Fanuc KAREL source: CA0044.KL

-- PROVISIONAL review KL for V770-1; original PC SHA256 f519f34b8b673ea591116af9cf0e5e1c5a1d14f930d2b18fb79fd747858d793d
-- Incomplete behavior may be omitted. Consult companion uncertainty JSON. Do not deploy.
PROGRAM CA0044
%NOLOCKGROUP
BEGIN
  -- UNRESOLVED_PC offsets 0-1; opcodes 7B
  -- UNRESOLVED_PC offsets 6-20; opcodes 21,9D,52,23
  -- UNRESOLVED_PC offsets 25-29; opcodes 7F
  -- UNRESOLVED_PC offsets 34-41; opcodes 9C,23
  -- UNRESOLVED_PC offsets 46-53; opcodes 9D,23
  -- UNRESOLVED_PC offsets 58-69; opcodes 2E,23
  -- UNRESOLVED_PC offsets 74-81; opcodes 9D,23
  -- UNRESOLVED_PC offsets 86-95; opcodes 3F,75
  -- UNRESOLVED_PC offsets 100-114; opcodes 2E,22,9D,33,35
  -- UNRESOLVED_PC offsets 119-133; opcodes 2E,22,9D,33,35
  -- UNRESOLVED_PC offsets 138-153; opcodes 2E,22,32,35
  -- UNRESOLVED_PC offsets 158-173; opcodes 2E,22,32,35
  -- UNRESOLVED_PC offsets 178-350; opcodes 27,27,21,27,21,27,21,27,21,27,21,27,21,27,21,27,21,27,21,27,21,27,21,27,21,27,21,27,21,27,21,27,21,27,21,27,21,27,21,27,21,27,21,27,21,27,21,27,21,AA
  -- UNRESOLVED_PC offsets 355-359; opcodes 7F
END CA0044
